      - frame TeachingPoints_07-17-05 at (8033.67, 5307.34, 828.56) mm, rotated rx 180 ry 0 rz 0 deg
        - target Point_07-17-05 (Cartesian target) at (0, 0, 0) mm; joints [8100, 12650, 655] of gantry
      - frame TeachingPoints_08-17-05 at (8733.67, 5307.34, 828.56) mm, rotated rx 180 ry 0 rz 0 deg
        - target Point_08-17-05 (Cartesian target) at (0, 0, 0) mm; joints [8800, 12650, 655] of gantry
      - frame TeachingPoints_09-17-05 at (9433.67, 5307.34, 828.56) mm, rotated rx 180 ry 0 rz 0 deg
        - target Point_09-17-05 (Cartesian target) at (0, 0, 0) mm; joints [9500, 12650, 655] of gantry
      - frame TeachingPoints_10-17-05 at (10133.67, 5307.34, 828.56) mm, rotated rx 180 ry 0 rz 0 deg
        - target Point_10-17-05 (Cartesian target) at (0, 0, 0) mm; joints [10200, 12650, 655] of gantry
      - frame TeachingPoints_11-17-05 at (10833.67, 5307.34, 828.56) mm, rotated rx 180 ry 0 rz 0 deg
        - target Point_11-17-05 (Cartesian target) at (0, 0, 0) mm; joints [10900, 12650, 655] of gantry
      - frame TeachingPoints_12-17-05 at (11533.67, 5307.34, 828.56) mm, rotated rx 180 ry 0 rz 0 deg
        - target Point_12-17-05 (Cartesian target) at (0, 0, 0) mm; joints [11600, 12650, 655] of gantry
      - frame TeachingPoints_13-17-05 at (12233.67, 5307.34, 828.56) mm, rotated rx 180 ry 0 rz 0 deg
        - target Point_13-17-05 (Cartesian target) at (0, 0, 0) mm; joints [12300, 12650, 655] of gantry
      - frame TeachingPoints_14-17-05 at (12933.67, 5307.34, 828.56) mm, rotated rx 180 ry 0 rz 0 deg
        - target Point_14-17-05 (Cartesian target) at (0, 0, 0) mm; joints [13000, 12650, 655] of gantry
      - frame TeachingPoints_15-17-05 at (13633.67, 5307.34, 828.56) mm, rotated rx 180 ry 0 rz 0 deg
        - target Point_15-17-05 (Cartesian target) at (0, 0, 0) mm; joints [13700, 12650, 655] of gantry
      - frame TeachingPoints_16-17-05 at (14333.67, 5307.34, 828.56) mm, rotated rx 180 ry 0 rz 0 deg
        - target Point_16-17-05 (Cartesian target) at (0, 0, 0) mm; joints [14400, 12650, 655] of gantry
      - frame TeachingPoints_17-17-05 at (15033.67, 5307.34, 828.56) mm, rotated rx 180 ry 0 rz 0 deg
        - target Point_17-17-05 (Cartesian target) at (0, 0, 0) mm; joints [15100, 12650, 655] of gantry
      - frame TeachingPoints_18-17-05 at (15733.67, 5307.34, 828.56) mm, rotated rx 180 ry 0 rz 0 deg
        - target Point_18-17-05 (Cartesian target) at (0, 0, 0) mm; joints [15800, 12650, 655] of gantry
      - frame TeachingPoints_19-17-05 at (16433.67, 5307.34, 828.56) mm, rotated rx 180 ry 0 rz 0 deg
        - target Point_19-17-05 (Cartesian target) at (0, 0, 0) mm; joints [16500, 12650, 655] of gantry
      - frame TeachingPoints_20-17-05 at (17133.67, 5307.34, 828.56) mm, rotated rx 180 ry 0 rz 0 deg
        - target Point_20-17-05 (Cartesian target) at (0, 0, 0) mm; joints [17200, 12650, 655] of gantry
      - frame TeachingPoints_01-18-05 at (3833.67, 4607.34, 828.56) mm, rotated rx 180 ry 0 rz 0 deg
        - target Point_01-18-05 (Cartesian target) at (0, 0, 0) mm; joints [3900, 13350, 655] of gantry
      - frame TeachingPoints_02-18-05 at (4533.67, 4607.34, 828.56) mm, rotated rx 180 ry 0 rz 0 deg
        - target Point_02-18-05 (Cartesian target) at (0, 0, 0) mm; joints [4600, 13350, 655] of gantry
      - frame TeachingPoints_03-18-05 at (5233.67, 4607.34, 828.56) mm, rotated rx 180 ry 0 rz 0 deg
        - target Point_03-18-05 (Cartesian target) at (0, 0, 0) mm; joints [5300, 13350, 655] of gantry
      - frame TeachingPoints_04-18-05 at (5933.67, 4607.34, 828.56) mm, rotated rx 180 ry 0 rz 0 deg
        - target Point_04-18-05 (Cartesian target) at (0, 0, 0) mm; joints [6000, 13350, 655] of gantry
      - frame TeachingPoints_05-18-05 at (6633.67, 4607.34, 828.56) mm, rotated rx 180 ry 0 rz 0 deg
        - target Point_05-18-05 (Cartesian target) at (0, 0, 0) mm; joints [6700, 13350, 655] of gantry
      - frame TeachingPoints_06-18-05 at (7333.67, 4607.34, 828.56) mm, rotated rx 180 ry 0 rz 0 deg
        - target Point_06-18-05 (Cartesian target) at (0, 0, 0) mm; joints [7400, 13350, 655] of gantry
      - frame TeachingPoints_07-18-05 at (8033.67, 4607.34, 828.56) mm, rotated rx 180 ry 0 rz 0 deg
        - target Point_07-18-05 (Cartesian target) at (0, 0, 0) mm; joints [8100, 13350, 655] of gantry
      - frame TeachingPoints_08-18-05 at (8733.67, 4607.34, 828.56) mm, rotated rx 180 ry 0 rz 0 deg
        - target Point_08-18-05 (Cartesian target) at (0, 0, 0) mm; joints [8800, 13350, 655] of gantry
      - frame TeachingPoints_09-18-05 at (9433.67, 4607.34, 828.56) mm, rotated rx 180 ry 0 rz 0 deg
        - target Point_09-18-05 (Cartesian target) at (0, 0, 0) mm; joints [9500, 13350, 655] of gantry
      - frame TeachingPoints_10-18-05 at (10133.67, 4607.34, 828.56) mm, rotated rx 180 ry 0 rz 0 deg
        - target Point_10-18-05 (Cartesian target) at (0, 0, 0) mm; joints [10200, 13350, 655] of gantry
      - frame TeachingPoints_11-18-05 at (10833.67, 4607.34, 828.56) mm, rotated rx 180 ry 0 rz 0 deg
        - target Point_11-18-05 (Cartesian target) at (0, 0, 0) mm; joints [10900, 13350, 655] of gantry
      - frame TeachingPoints_12-18-05 at (11533.67, 4607.34, 828.56) mm, rotated rx 180 ry 0 rz 0 deg
        - target Point_12-18-05 (Cartesian target) at (0, 0, 0) mm; joints [11600, 13350, 655] of gantry
      - frame TeachingPoints_13-18-05 at (12233.67, 4607.34, 828.56) mm, rotated rx 180 ry 0 rz 0 deg
        - target Point_13-18-05 (Cartesian target) at (0, 0, 0) mm; joints [12300, 13350, 655] of gantry
      - frame TeachingPoints_14-18-05 at (12933.67, 4607.34, 828.56) mm, rotated rx 180 ry 0 rz 0 deg
        - target Point_14-18-05 (Cartesian target) at (0, 0, 0) mm; joints [13000, 13350, 655] of gantry
      - frame TeachingPoints_15-18-05 at (13633.67, 4607.34, 828.56) mm, rotated rx 180 ry 0 rz 0 deg
        - target Point_15-18-05 (Cartesian target) at (0, 0, 0) mm; joints [13700, 13350, 655] of gantry
      - frame TeachingPoints_16-18-05 at (14333.67, 4607.34, 828.56) mm, rotated rx 180 ry 0 rz 0 deg
        - target Point_16-18-05 (Cartesian target) at (0, 0, 0) mm; joints [14400, 13350, 655] of gantry
      - frame TeachingPoints_17-18-05 at (15033.67, 4607.34, 828.56) mm, rotated rx 180 ry 0 rz 0 deg
        - target Point_17-18-05 (Cartesian target) at (0, 0, 0) mm; joints [15100, 13350, 655] of gantry
      - frame TeachingPoints_18-18-05 at (15733.67, 4607.34, 828.56) mm, rotated rx 180 ry 0 rz 0 deg
        - target Point_18-18-05 (Cartesian target) at (0, 0, 0) mm; joints [15800, 13350, 655] of gantry
      - frame TeachingPoints_19-18-05 at (16433.67, 4607.34, 828.56) mm, rotated rx 180 ry 0 rz 0 deg
        - target Point_19-18-05 (Cartesian target) at (0, 0, 0) mm; joints [16500, 13350, 655] of gantry
      - frame TeachingPoints_20-18-05 at (17133.67, 4607.34, 828.56) mm, rotated rx 180 ry 0 rz 0 deg
        - target Point_20-18-05 (Cartesian target) at (0, 0, 0) mm; joints [17200, 13350, 655] of gantry
      - frame TeachingPoints_01-19-05 at (3833.67, 3907.34, 828.56) mm, rotated rx 180 ry 0 rz 0 deg
        - target Point_01-19-05 (Cartesian target) at (0, 0, 0) mm; joints [3900, 14050, 655] of gantry
      - frame TeachingPoints_02-19-05 at (4533.67, 3907.34, 828.56) mm, rotated rx 180 ry 0 rz 0 deg
        - target Point_02-19-05 (Cartesian target) at (0, 0, 0) mm; joints [4600, 14050, 655] of gantry
      - frame TeachingPoints_03-19-05 at (5233.67, 3907.34, 828.56) mm, rotated rx 180 ry 0 rz 0 deg
        - target Point_03-19-05 (Cartesian target) at (0, 0, 0) mm; joints [5300, 14050, 655] of gantry
      - frame TeachingPoints_04-19-05 at (5933.67, 3907.34, 828.56) mm, rotated rx 180 ry 0 rz 0 deg
        - target Point_04-19-05 (Cartesian target) at (0, 0, 0) mm; joints [6000, 14050, 655] of gantry
      - frame TeachingPoints_05-19-05 at (6633.67, 3907.34, 828.56) mm, rotated rx 180 ry 0 rz 0 deg
        - target Point_05-19-05 (Cartesian target) at (0, 0, 0) mm; joints [6700, 14050, 655] of gantry
      - frame TeachingPoints_06-19-05 at (7333.67, 3907.34, 828.56) mm, rotated rx 180 ry 0 rz 0 deg
        - target Point_06-19-05 (Cartesian target) at (0, 0, 0) mm; joints [7400, 14050, 655] of gantry
      - frame TeachingPoints_07-19-05 at (8033.67, 3907.34, 828.56) mm, rotated rx 180 ry 0 rz 0 deg
        - target Point_07-19-05 (Cartesian target) at (0, 0, 0) mm; joints [8100, 14050, 655] of gantry
      - frame TeachingPoints_08-19-05 at (8733.67, 3907.34, 828.56) mm, rotated rx 180 ry 0 rz 0 deg
        - target Point_08-19-05 (Cartesian target) at (0, 0, 0) mm; joints [8800, 14050, 655] of gantry
      - frame TeachingPoints_09-19-05 at (9433.67, 3907.34, 828.56) mm, rotated rx 180 ry 0 rz 0 deg
        - target Point_09-19-05 (Cartesian target) at (0, 0, 0) mm; joints [9500, 14050, 655] of gantry
      - frame TeachingPoints_10-19-05 at (10133.67, 3907.34, 828.56) mm, rotated rx 180 ry 0 rz 0 deg
        - target Point_10-19-05 (Cartesian target) at (0, 0, 0) mm; joints [10200, 14050, 655] of gantry
      - frame TeachingPoints_11-19-05 at (10833.67, 3907.34, 828.56) mm, rotated rx 180 ry 0 rz 0 deg
        - target Point_11-19-05 (Cartesian target) at (0, 0, 0) mm; joints [10900, 14050, 655] of gantry
      - frame TeachingPoints_12-19-05 at (11533.67, 3907.34, 828.56) mm, rotated rx 180 ry 0 rz 0 deg
        - target Point_12-19-05 (Cartesian target) at (0, 0, 0) mm; joints [11600, 14050, 655] of gantry
      - frame TeachingPoints_13-19-05 at (12233.67, 3907.34, 828.56) mm, rotated rx 180 ry 0 rz 0 deg
        - target Point_13-19-05 (Cartesian target) at (0, 0, 0) mm; joints [12300, 14050, 655] of gantry
      - frame TeachingPoints_14-19-05 at (12933.67, 3907.34, 828.56) mm, rotated rx 180 ry 0 rz 0 deg
        - target Point_14-19-05 (Cartesian target) at (0, 0, 0) mm; joints [13000, 14050, 655] of gantry
      - frame TeachingPoints_15-19-05 at (13633.67, 3907.34, 828.56) mm, rotated rx 180 ry 0 rz 0 deg
        - target Point_15-19-05 (Cartesian target) at (0, 0, 0) mm; joints [13700, 14050, 655] of gantry
      - frame TeachingPoints_16-19-05 at (14333.67, 3907.34, 828.56) mm, rotated rx 180 ry 0 rz 0 deg
        - target Point_16-19-05 (Cartesian target) at (0, 0, 0) mm; joints [14400, 14050, 655] of gantry
      - frame TeachingPoints_17-19-05 at (15033.67, 3907.34, 828.56) mm, rotated rx 180 ry 0 rz 0 deg
        - target Point_17-19-05 (Cartesian target) at (0, 0, 0) mm; joints [15100, 14050, 655] of gantry
      - frame TeachingPoints_18-19-05 at (15733.67, 3907.34, 828.56) mm, rotated rx 180 ry 0 rz 0 deg
        - target Point_18-19-05 (Cartesian target) at (0, 0, 0) mm; joints [15800, 14050, 655] of gantry
      - frame TeachingPoints_19-19-05 at (16433.67, 3907.34, 828.56) mm, rotated rx 180 ry 0 rz 0 deg
        - target Point_19-19-05 (Cartesian target) at (0, 0, 0) mm; joints [16500, 14050, 655] of gantry
      - frame TeachingPoints_20-19-05 at (17133.67, 3907.34, 828.56) mm, rotated rx 180 ry 0 rz 0 deg
        - target Point_20-19-05 (Cartesian target) at (0, 0, 0) mm; joints [17200, 14050, 655] of gantry
      - frame TeachingPoints_01-20-05 at (3833.67, 3207.34, 828.56) mm, rotated rx 180 ry 0 rz 0 deg
        - target Point_01-20-05 (Cartesian target) at (0, 0, 0) mm; joints [3900, 14750, 655] of gantry
      - frame TeachingPoints_02-20-05 at (4533.67, 3207.34, 828.56) mm, rotated rx 180 ry 0 rz 0 deg
        - target Point_02-20-05 (Cartesian target) at (0, 0, 0) mm; joints [4600, 14750, 655] of gantry
      - frame TeachingPoints_03-20-05 at (5233.67, 3207.34, 828.56) mm, rotated rx 180 ry 0 rz 0 deg
        - target Point_03-20-05 (Cartesian target) at (0, 0, 0) mm; joints [5300, 14750, 655] of gantry
      - frame TeachingPoints_04-20-05 at (5933.67, 3207.34, 828.56) mm, rotated rx 180 ry 0 rz 0 deg
        - target Point_04-20-05 (Cartesian target) at (0, 0, 0) mm; joints [6000, 14750, 655] of gantry
      - frame TeachingPoints_05-20-05 at (6633.67, 3207.34, 828.56) mm, rotated rx 180 ry 0 rz 0 deg
        - target Point_05-20-05 (Cartesian target) at (0, 0, 0) mm; joints [6700, 14750, 655] of gantry
      - frame TeachingPoints_06-20-05 at (7333.67, 3207.34, 828.56) mm, rotated rx 180 ry 0 rz 0 deg
        - target Point_06-20-05 (Cartesian target) at (0, 0, 0) mm; joints [7400, 14750, 655] of gantry
      - frame TeachingPoints_07-20-05 at (8033.67, 3207.34, 828.56) mm, rotated rx 180 ry 0 rz 0 deg
        - target Point_07-20-05 (Cartesian target) at (0, 0, 0) mm; joints [8100, 14750, 655] of gantry
      - frame TeachingPoints_08-20-05 at (8733.67, 3207.34, 828.56) mm, rotated rx 180 ry 0 rz 0 deg
        - target Point_08-20-05 (Cartesian target) at (0, 0, 0) mm; joints [8800, 14750, 655] of gantry
      - frame TeachingPoints_09-20-05 at (9433.67, 3207.34, 828.56) mm, rotated rx 180 ry 0 rz 0 deg
        - target Point_09-20-05 (Cartesian target) at (0, 0, 0) mm; joints [9500, 14750, 655] of gantry
      - frame TeachingPoints_10-20-05 at (10133.67, 3207.34, 828.56) mm, rotated rx 180 ry 0 rz 0 deg
        - target Point_10-20-05 (Cartesian target) at (0, 0, 0) mm; joints [10200, 14750, 655] of gantry
      - frame TeachingPoints_11-20-05 at (10833.67, 3207.34, 828.56) mm, rotated rx 180 ry 0 rz 0 deg
        - target Point_11-20-05 (Cartesian target) at (0, 0, 0) mm; joints [10900, 14750, 655] of gantry
      - frame TeachingPoints_12-20-05 at (11533.67, 3207.34, 828.56) mm, rotated rx 180 ry 0 rz 0 deg
        - target Point_12-20-05 (Cartesian target) at (0, 0, 0) mm; joints [11600, 14750, 655] of gantry
      - frame TeachingPoints_13-20-05 at (12233.67, 3207.34, 828.56) mm, rotated rx 180 ry 0 rz 0 deg
        - target Point_13-20-05 (Cartesian target) at (0, 0, 0) mm; joints [12300, 14750, 655] of gantry
      - frame TeachingPoints_14-20-05 at (12933.67, 3207.34, 828.56) mm, rotated rx 180 ry 0 rz 0 deg
        - target Point_14-20-05 (Cartesian target) at (0, 0, 0) mm; joints [13000, 14750, 655] of gantry
      - frame TeachingPoints_15-20-05 at (13633.67, 3207.34, 828.56) mm, rotated rx 180 ry 0 rz 0 deg
        - target Point_15-20-05 (Cartesian target) at (0, 0, 0) mm; joints [13700, 14750, 655] of gantry
      - frame TeachingPoints_16-20-05 at (14333.67, 3207.34, 828.56) mm, rotated rx 180 ry 0 rz 0 deg
        - target Point_16-20-05 (Cartesian target) at (0, 0, 0) mm; joints [14400, 14750, 655] of gantry
      - frame TeachingPoints_17-20-05 at (15033.67, 3207.34, 828.56) mm, rotated rx 180 ry 0 rz 0 deg
        - target Point_17-20-05 (Cartesian target) at (0, 0, 0) mm; joints [15100, 14750, 655] of gantry
      - frame TeachingPoints_18-20-05 at (15733.67, 3207.34, 828.56) mm, rotated rx 180 ry 0 rz 0 deg
        - target Point_18-20-05 (Cartesian target) at (0, 0, 0) mm; joints [15800, 14750, 655] of gantry
      - frame TeachingPoints_19-20-05 at (16433.67, 3207.34, 828.56) mm, rotated rx 180 ry 0 rz 0 deg
        - target Point_19-20-05 (Cartesian target) at (0, 0, 0) mm; joints [16500, 14750, 655] of gantry
      - frame TeachingPoints_20-20-05 at (17133.67, 3207.34, 828.56) mm, rotated rx 180 ry 0 rz 0 deg
        - target Point_20-20-05 (Cartesian target) at (0, 0, 0) mm; joints [17200, 14750, 655] of gantry
